{attribute 'qualified_only'}
VAR_GLOBAL
	FwLimit				AT	%I*	: ARRAY[1..GVL.axisNumMax] OF BOOL;
	BwLimit				AT  %I*	: ARRAY[1..GVL.axisNumMax] OF BOOL;
	
	FwLimitsCoupling	: ARRAY [1..GVL.axisNumMax] OF ARRAY [1..GVL.axisNumMax] OF limitCoupling;
	BwLimitsCoupling	: ARRAY [1..GVL.axisNumMax] OF ARRAY [1..GVL.axisNumMax] OF limitCoupling;

	
END_VAR

(* stored: Version 1.1.0.1, ProductVersion 3.1.4020.12
   GVL Limits: Id {bc15940f-38e2-463e-88a6-afd29e0a1edc} *)
